{attribute addProperty BoxType "EL1502--0000"}
{attribute addProperty Id "Output_functions_enabledAT %I*BOOL811Status_of_outputAT %I*BOOL812Set_counter_doneAT %I*BOOL813Counter_inhibitedAT %I*BOOL814Status_of_input_UDAT %I*BOOL815Status_of_input_clockAT %I*BOOL816TxPDO_ToggleAT %I*BOOL819Counter_valueAT %I*UDINT32417"}
{attribute addProperty CRC "768713232"}
{attribute addProperty SizeInBites "88"}
{attribute addProperty SizeInBytes "11"}
TYPE CNT_Inputs_2DD1A210 :
STRUCT
	{attribute addProperty Name "Output_functions_enabled"}
	Output_functions_enabled AT %I* : BOOL;
	{attribute addProperty Name "Status_of_output"}
	Status_of_output AT %I* : BOOL;
	{attribute addProperty Name "Set_counter_done"}
	Set_counter_done AT %I* : BOOL;
	{attribute addProperty Name "Counter_inhibited"}
	Counter_inhibited AT %I* : BOOL;
	{attribute addProperty Name "Status_of_input_UD"}
	Status_of_input_UD AT %I* : BOOL;
	{attribute addProperty Name "Status_of_input_clock"}
	Status_of_input_clock AT %I* : BOOL;
	{attribute addProperty Name "TxPDO_Toggle"}
	TxPDO_Toggle AT %I* : BOOL;
	{attribute addProperty Name "Counter_value"}
	Counter_value AT %I* : UDINT;
END_STRUCT
END_TYPE

(* stored: Version 1.2.0.0, ProductVersion 3.1.4024.9
   DUT CNT_Inputs_2DD1A210: Id {3ae35ad6-2105-45c7-932a-404dcdcceb19} *)
